(* CODESYS project Soru_3.project
   Title: Adsız2
   Version: 0.0.0.0
   Author: Enes

Project tree, tasks and I/O mapping:
  MyController : TM241C24T/U, Schneider Electric, order no. TM241C24T/U, version 4.0.6.18
    application Application
      task MAST (cyclic, interval 20 ms, priority 15, watchdog 100 ms x 1) calls POU
      global variables GVL
      program POU [LD]
    DI : Digital Inputs, Schneider Electric, version 4.0.6.18
        input  iwDI_IW0 : WORD  // IW0
        input  ibDI_IB1 : BYTE  // IB1
    DQ : Digital Outputs, Schneider Electric, version 4.0.6.18
        output qwDQ_QW0 : WORD  // QW0
        output qbDQ_QB1 : BYTE  // QB1
    Counters : Counters, Schneider Electric, version 4.0.6.18
    Pulse_Generators : Pulse Generators, Schneider Electric, version 4.0.6.18
    Cartridge_1 : Cartridge, Schneider Electric, version 4.0.6.18
    IO_Bus : IO bus - TM3, Schneider Electric, version 4.0.6.18
    COM_Bus : COM bus, Schneider Electric, version 4.0.6.18
    Serial_Line_1 : Serial line, Schneider Electric, version 4.0.6.18
      SoMachine_Network_Manager : SoMachine-Network Manager, Schneider Electric, version 4.0.0.2
    Serial_Line_2 : Serial line, Schneider Electric, version 4.0.6.18
      Modbus_Manager : Modbus Manager, Schneider Electric, version 4.0.0.2
*)

// MyController/Application/GVL
VAR_GLOBAL
END_VAR

// MyController/Application/POU
PROGRAM POU
VAR
	Start: BOOL;
	Stop: BOOL;
	M0: BOOL;
	Motor_1: BOOL;
	Timer1: TON;
	Motor_2: BOOL;
	Timer3: TON;
	Motor1_Asiri_Akim: BOOL;
	Motor2_Asiri_Akim: BOOL;
END_VAR

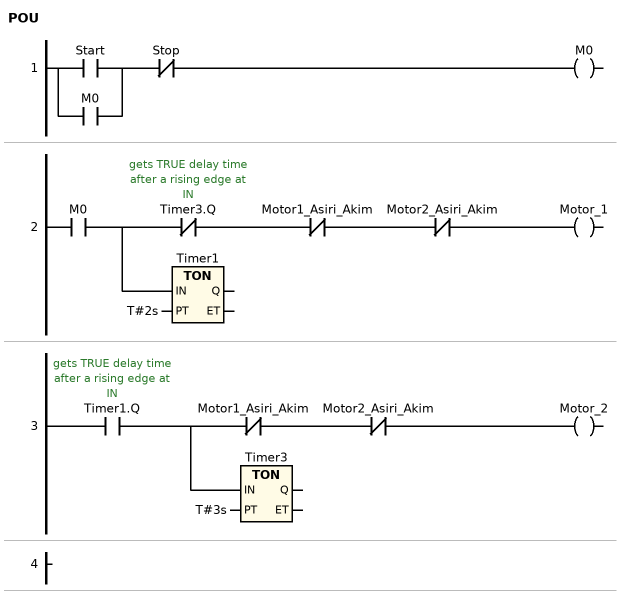
// NETWORK 1
M0 := (Start OR M0) AND NOT Stop;

// NETWORK 2
//   Timer3.Q: gets TRUE delay time after a rising edge at IN
Motor_1 := M0 AND NOT Timer3.Q AND NOT Motor1_Asiri_Akim AND NOT Motor2_Asiri_Akim;
Timer1(IN := M0, PT := T#2s); // TON

// NETWORK 3
//   Timer1.Q: gets TRUE delay time after a rising edge at IN
Motor_2 := Timer1.Q AND NOT Motor1_Asiri_Akim AND NOT Motor2_Asiri_Akim;
Timer3(IN := Timer1.Q, PT := T#3s); // TON

// NETWORK 4

END_PROGRAM
